TYPE DUT_HMI_Events :
STRUCT
	Clear :BOOL;
END_STRUCT
END_TYPE

(* stored: Version 1.1.0.1, ProductVersion 3.1.4024.13
   DUT DUT_HMI_Events: Id {eb89f784-c887-4283-abb5-68cb7d870607} *)
